// TIA Portal project "Konvenyör Bandını Hızlandırma Ve Yavaşlatma Çalışması_V15.1" (V15.1)
// Vorlageprojekt für das Buch mit Zielsystem S7-1200

(* hardware
DEVICE "S7-1200-Station_1"  S7-1200 Station
   slot 0: "Baugruppenträger_0"  Rack  V1.0
   slot 1: "PLC_1"  CPU 1211C DC/DC/DC  6ES7 211-1AE40-0XB0  V4.1
DEVICE "PC-System_1"  SIMATIC PC station
   slot 0: "SIMATIC PC station"  Rail  SIMATIC PC-Station  V1.0
      slot 125: "Stationmanager"  Station_Manager  V6.0.4
   slot 1: "HMI_RT_1"  WinCC RT Advanced  6AV2 104-0xxxx-xxxx  15.1.0.0
      slot 33792: "Host interface"  Host interface
   slot 2: "IE general_1"  IE General  IE_CP  V8.2.0
*)

// ===== PLC "PLC_1"  CPU 1211C DC/DC/DC =====

VAR_GLOBAL   // PLC tag table "plc_tags"
   "stop" AT %I0.0 : Bool;
   "start" AT %I0.1 : Bool;
   "sistem_devrede" AT %M5.0 : Bool;
   "st_mem" AT %M5.1 : Bool;
   "hızlandir_butonu" AT %I0.2 : Bool;
   "yükselen kenar" AT %M5.3 : Bool;
   "hizlandirma_siddeti" AT %QW32 : Int;
   "konvenyor_hizi" AT %QW30 : Int;
   "konvenyor_Devrede_lambasi" AT %Q0.1 : Bool;
   "konvenyor_stop_lambası" AT %Q0.2 : Bool;
END_VAR

VAR_GLOBAL   // PLC tag table "hmi_tags"
   "hmi_start" AT %M6.0 : Bool;
   "hmi_stop" AT %M6.1 : Bool;
   "hmi_hızlandir" AT %M6.2 : Bool;
END_VAR

// folder: System blocks/Program resources

DATA_BLOCK "hızlandırma_seviyesi_kontrol_sayaci"   // DB1
{ S7_Optimized_Access := 'TRUE' }
AUTHOR : Simatic
FAMILY : IEC
NAME : CNTR
VERSION : 1.0
// stored: InstanceOfName IEC_COUNTER
"IEC_COUNTER"
BEGIN
END_DATA_BLOCK

// folder: (top level)

FUNCTION "MHJ-PLC-Lab-Function-S71200" : Void   // FC9000, SCL
{ S7_Optimized_Access := 'TRUE' }
VERSION : 0.1
   VAR_TEMP
      rdTimeReturn : Int;
      outputTime : DTL;
      SyncVal : Byte;
      forVal : Int;
      forVal_2 : Int;
      Value : Byte;
   END_VAR
   VAR CONSTANT
      CompVal : Byte := 16#34;
      Value_01 : Byte := 16#11;
      Value_01_DW : DWord := 16#A165_D992;
      Value_02_DW : DWord := 16#58BE_4401;
   END_VAR
BEGIN

   #Value:=PEEK(area := 16#82,
        dbNumber := 0,
        byteOffset := 511);
   #Value := #Value + 1;

   POKE(area := 16#82,
        dbNumber := 0,
        byteOffset := 511,
        value := #Value);

   POKE(area:=16#81,
        dbNumber:=0,
        byteOffset:=1016,
        value:=#Value_01_DW);
   POKE(area := 16#81,
        dbNumber := 0,
        byteOffset := 1020,
        value := #Value_02_DW);

   POKE(area := 16#81,
        dbNumber := 0,
        byteOffset := 511,
        value := B#16#00);

   FOR #forVal := 0 TO 120 DO
       FOR #forVal_2:=0 TO 10 DO
           #rdTimeReturn:=RD_SYS_T(#outputTime);
           #rdTimeReturn := WR_SYS_T(#outputTime);
           #rdTimeReturn := RD_SYS_T(#outputTime);
           #rdTimeReturn := WR_SYS_T(#outputTime);
       END_FOR;
       #SyncVal:= PEEK(area := 16#81,
                      dbNumber := 0,
                      byteOffset := 511);
       IF #SyncVal = #CompVal THEN
          GOTO M_1;
       END_IF;
   END_FOR;
   RETURN;

   M_1:
   POKE(area := 16#81,
        dbNumber := 0,
        byteOffset := 511,
        value := B#16#0);
END_FUNCTION

ORGANIZATION_BLOCK "Main"   // OB1, LAD, ProgramCycle
TITLE = "Main Program Sweep (Cycle)"
{ S7_Optimized_Access := 'TRUE' }
VERSION : 0.1
   VAR_INPUT
      Initial_Call : Bool;   // Initial call of this OB
      Remanence : Bool;   // =True, if remanent data are available
   END_VAR
   VAR_TEMP
      konvenyör_hizi : Int;
   END_VAR
   VAR_TEMP   // added for the SCL form of the ladder/FBD networks
      _w1 : Bool;
      _w2 : Bool;
   END_VAR
BEGIN

REGION Network 1: Konnektierungsbaustein für PLC-Lab
   // Im Netzwerk 1 wird der Konnektierungsbaustein für PLC-Lab aufgerufen.
   // Dieser Aufruf darf nicht entfernt werden!
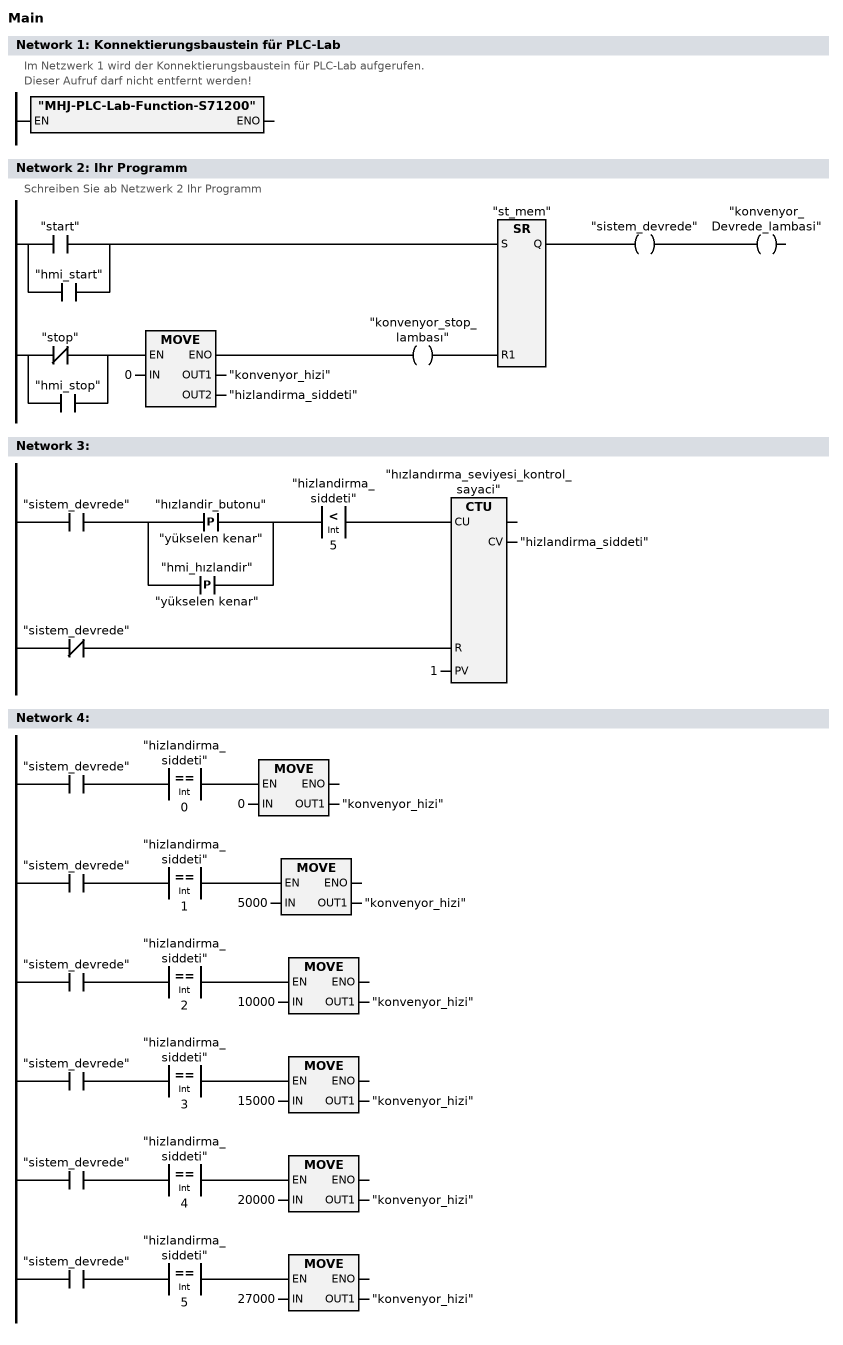
   RUNG wire#powerrail
      "MHJ-PLC-Lab-Function-S71200"()
   END_RUNG
   // the same network as SCL:
   "MHJ-PLC-Lab-Function-S71200"();
END_REGION

REGION Network 2: Ihr Programm
   // Schreiben Sie ab Netzwerk 2 Ihr Programm
   RUNG wire#powerrail
      Contact( "start" )
      wire#w1
      S_SR(operand := "st_mem", r1 := wire#w3)
      Coil( "sistem_devrede" )
      Coil( "konvenyor_Devrede_lambasi" )
   END_RUNG
   RUNG wire#powerrail
      Contact( "hmi_start" )
   END_RUNG wire#w1
   RUNG wire#powerrail
      I_Contact( "stop" )
      wire#w2
      Move(in := 0, out1 => "konvenyor_hizi", out2 => "hizlandirma_siddeti")
      Coil( "konvenyor_stop_lambası" )
   END_RUNG wire#w3
   RUNG wire#powerrail
      Contact( "hmi_stop" )
   END_RUNG wire#w2
   // the same network as SCL:
   #_w1 := NOT "stop" OR "hmi_stop";
   IF #_w1 THEN
       "konvenyor_hizi" := 0;
       "hizlandirma_siddeti" := 0;
   END_IF;
   "konvenyor_stop_lambası" := #_w1;
   IF "start" OR "hmi_start" THEN
       "st_mem" := TRUE;   // SR flip-flop
   END_IF;
   IF #_w1 THEN "st_mem" := FALSE; END_IF;
   "sistem_devrede" := "st_mem";
   "konvenyor_Devrede_lambasi" := "st_mem";
END_REGION

REGION Network 3
   #_w1 := "sistem_devrede" AND "hızlandir_butonu" AND NOT "yükselen kenar";   // rising edge of "hızlandir_butonu"
   "yükselen kenar" := "hızlandir_butonu";
   #_w2 := "sistem_devrede" AND "hmi_hızlandir" AND NOT "yükselen kenar";   // rising edge of "hmi_hızlandir"
   "yükselen kenar" := "hmi_hızlandir";
   "hızlandırma_seviyesi_kontrol_sayaci".CTU(CU := (#_w1 OR #_w2) AND ("hizlandirma_siddeti" < 5),
                           R := NOT "sistem_devrede",
                           PV := 1,
                           CV => "hizlandirma_siddeti");
END_REGION

REGION Network 4
   RUNG wire#powerrail
      Contact( "sistem_devrede" )
      { S7_Templates := "SrcType := Int" } EQ_Contact(in1 := "hizlandirma_siddeti", in2 := 0)
      Move(in := 0, out1 => "konvenyor_hizi")
   END_RUNG
   RUNG wire#powerrail
      Contact( "sistem_devrede" )
      { S7_Templates := "SrcType := Int" } EQ_Contact(in1 := "hizlandirma_siddeti", in2 := 1)
      Move(in := 5000, out1 => "konvenyor_hizi")
   END_RUNG
   RUNG wire#powerrail
      Contact( "sistem_devrede" )
      { S7_Templates := "SrcType := Int" } EQ_Contact(in1 := "hizlandirma_siddeti", in2 := 2)
      Move(in := 10000, out1 => "konvenyor_hizi")
   END_RUNG
   RUNG wire#powerrail
      Contact( "sistem_devrede" )
      { S7_Templates := "SrcType := Int" } EQ_Contact(in1 := "hizlandirma_siddeti", in2 := 3)
      Move(in := 15000, out1 => "konvenyor_hizi")
   END_RUNG
   RUNG wire#powerrail
      Contact( "sistem_devrede" )
      { S7_Templates := "SrcType := Int" } EQ_Contact(in1 := "hizlandirma_siddeti", in2 := 4)
      Move(in := 20000, out1 => "konvenyor_hizi")
   END_RUNG
   RUNG wire#powerrail
      Contact( "sistem_devrede" )
      { S7_Templates := "SrcType := Int" } EQ_Contact(in1 := "hizlandirma_siddeti", in2 := 5)
      Move(in := 27000, out1 => "konvenyor_hizi")
   END_RUNG
   // the same network as SCL:
   IF "sistem_devrede" AND ("hizlandirma_siddeti" = 0) THEN "konvenyor_hizi" := 0; END_IF;
   IF "sistem_devrede" AND ("hizlandirma_siddeti" = 1) THEN "konvenyor_hizi" := 5000; END_IF;
   IF "sistem_devrede" AND ("hizlandirma_siddeti" = 2) THEN "konvenyor_hizi" := 10000; END_IF;
   IF "sistem_devrede" AND ("hizlandirma_siddeti" = 3) THEN "konvenyor_hizi" := 15000; END_IF;
   IF "sistem_devrede" AND ("hizlandirma_siddeti" = 4) THEN "konvenyor_hizi" := 20000; END_IF;
   IF "sistem_devrede" AND ("hizlandirma_siddeti" = 5) THEN "konvenyor_hizi" := 27000; END_IF;
END_REGION
END_ORGANIZATION_BLOCK

(* ===== HMI "HMI_RT_1" =====
system functions are stored by id; their names below are inferred from use
connection "HMI_Connection_1": ETHERNET, S7_1200_OMS

HMI tags "Default tag table"
   "hmi_stop" : Bool = PLC hmi_stop AT %M6.1, 1 s
   "hmi_start" : Bool = PLC hmi_start AT %M6.0, 1 s
   "hmi_hızlandir" : Bool = PLC hmi_hızlandir AT %M6.2, 1 s
   "konvenyor_hizi" : Int = PLC konvenyor_hizi AT %QW30, 1 s
   "sistem_devrede" : Bool = PLC sistem_devrede AT %M5.0, 1 s

screen "Screen_1" 640x480
   Button "Button_1" at 75,190 size 96x32; TextOff 'START'
      on Press: SetBit("hmi_start")
      on Release: ResetBit("hmi_start")
   Button "Button_2" at 75,255 size 96x32; TextOff 'STOP'
      on Press: SetBit("hmi_stop")
      on Release: ResetBit("hmi_stop")
   Button "Button_3" at 96,319 size 50x45; TextOff 'HIZI AYARLA'
      on Press: SetBit("hmi_hızlandir")
      on Release: ResetBit("hmi_hızlandir")
   GraphicView "Graphic view_2" at 206,168 size 300x300; Picture "Graphic_2"
   GraphicView "Graphic view_3" at 249,295 size 215x184; Picture "Graphic_3"
   Circle "Circle_1" at 301,348 size 49x49
      Appearance <- "sistem_devrede"
   Circle "Circle_2" at 362,347 size 49x49
      Appearance <- "sistem_devrede"
   GraphicIOField "Graphic I/O field_1" at 415,102 size 96x48
      Appearance <- "konvenyor_hizi"
      ProcessValue <- "konvenyor_hizi"
*)